PROGRAM MAIN
VAR
	doSomething_instance1: DoSomething;
	
END_VAR

doSomething_instance1.method1();
doSomething_instance1(input := true);

END_PROGRAM

(* stored: Version 1.1.0.1, ProductVersion 3.1.4024.12
   POU MAIN: Id {50d6cc32-61c7-417e-bf3e-2120b9229e9c}, SpecialFunc None *)
